FUNCTION SetMat7_3 :  ARRAY [0..6,0..2] OF int
VAR_INPUT
	x_11:INT;
	x_12:INT;
	x_13:INT;
	x_21:INT;
	x_22:INT;
	x_23:INT;
	x_31:INT;
	x_32:INT;
	x_33:INT;
	x_41:INT;
	x_42:INT;
	x_43:INT;
	x_51:INT;
	x_52:INT;
	x_53:INT;
	x_61:INT;
	x_62:INT;
	x_63:INT;
	x_71:INT;
	x_72:INT;
	x_73:INT;
END_VAR
VAR_OUTPUT
END_VAR
VAR
END_VAR

SetMat7_3 [0,0]:=x_11;
SetMat7_3 [0,1]:=x_12;
SetMat7_3 [0,2]:=x_13;

SetMat7_3 [1,0]:=x_21;
SetMat7_3 [1,1]:=x_22;
SetMat7_3 [1,2]:=x_23;

SetMat7_3 [2,0]:=x_31;
SetMat7_3 [2,1]:=x_32;
SetMat7_3 [2,2]:=x_33;

SetMat7_3 [3,0]:=x_41;
SetMat7_3 [3,1]:=x_42;
SetMat7_3 [3,2]:=x_43;

SetMat7_3 [4,0]:=x_51;
SetMat7_3 [4,1]:=x_52;
SetMat7_3 [4,2]:=x_53;

SetMat7_3 [5,0]:=x_61;
SetMat7_3 [5,1]:=x_62;
SetMat7_3 [5,2]:=x_63;

SetMat7_3 [6,0]:=x_71;
SetMat7_3 [6,1]:=x_72;
SetMat7_3 [6,2]:=x_73;

END_FUNCTION

(* stored: Version 1.1.0.1, ProductVersion 3.1.4024.2
   POU SetMat7_3: Id {e70132cd-18c1-4604-8ee6-eb3f82adadab}, SpecialFunc None *)
